TYPE csp_transfer_upstacker_phase_status_enum :
(		
	CSP_TRANSFER_UPSTACKER_STATUS_PHASE_START								:= 0,
	CSP_TRANSFER_UPSTACKER_STATUS_PHASE_CHECK_VM_STATUS						:= 1,
	CSP_TRANSFER_UPSTACKER_STATUS_PHASE_GET_VM_POS							:= 2,
	CSP_TRANSFER_UPSTACKER_STATUS_PHASE_CALCULATE_SLAVE_POS					:= 3,
	CSP_TRANSFER_UPSTACKER_STATUS_PHASE_CALCULATE_SLAVE_DOWN_POS			:= 600,
	CSP_TRANSFER_UPSTACKER_STATUS_PHASE_CHECK_CALCULATED_SLAVE_DOWN_POS		:= 601,
	CSP_TRANSFER_UPSTACKER_STATUS_PHASE_CALCULATE_SLAVE_UP_POS				:= 602,
	CSP_TRANSFER_UPSTACKER_STATUS_PHASE_CHECK_CALCULATED_SLAVE_UP_POS		:= 603,
	CSP_TRANSFER_UPSTACKER_STATUS_PHASE_CALCULATE_SLAVE_LS_FINGER_POS		:= 604,
	CSP_TRANSFER_UPSTACKER_STATUS_PHASE_CHECK_CALCULATED_SLAVE_LSFINGR_POS	:= 605,
	CSP_TRANSFER_UPSTACKER_STATUS_PHASE_CALCULATE_SLAVE_OS_FINGER_POS		:= 606,
	CSP_TRANSFER_UPSTACKER_STATUS_PHASE_CHECK_CALCULATED_SLAVE_OSFINGR_POS	:= 607,
	CSP_TRANSFER_UPSTACKER_STATUS_PHASE_CHECK_SLAVE_POS						:= 4,
	CSP_TRANSFER_UPSTACKER_STATUS_PHASE_SIMPLE_MOVE_AVAILABLE				:= 5,
	CSP_TRANSFER_UPSTACKER_STATUS_PHASE_CALCULATE_IDLE_POSITION				:= 10,
	CSP_TRANSFER_UPSTACKER_STATUS_PHASE_REDEFINE_IDLE_POSITION				:= 15,
	CSP_TRANSFER_UPSTACKER_STATUS_PHASE_READ_IDLE_POSITION					:= 20,
	CSP_TRANSFER_UPSTACKER_STATUS_PHASE_CALCULATE_SLAVE_POSITION			:= 30,
	CSP_TRANSFER_UPSTACKER_STATUS_PHASE_READ_SLAVE_POSITION					:= 40,
	CSP_TRANSFER_UPSTACKER_STATUS_PHASE_CALCULATE_VIRTUAL_POSITION			:= 50,
	CSP_TRANSFER_UPSTACKER_STATUS_PHASE_READ_VIRTUAL_POSITION				:= 60,
	CSP_TRANSFER_UPSTACKER_STATUS_PHASE_CHECK_CASE							:= 70,
	CSP_TRANSFER_UPSTACKER_STATUS_PHASE_DISABLE 							:= 80,
	CSP_TRANSFER_UPSTACKER_STATUS_PHASE_ENABLE 								:= 90,
	CSP_TRANSFER_UPSTACKER_STATUS_PHASE_ENABLED								:= 100,
	CSP_TRANSFER_UPSTACKER_STATUS_PHASE_CHECK_UPSTREAM_SKIP_PHASING			:= 101,
	CSP_TRANSFER_UPSTACKER_STATUS_PHASE_CHECK_DOWNSTREAM_SKIP_PHASE_1		:= 110,
	CSP_TRANSFER_UPSTACKER_STATUS_PHASE_CALCULATE_MASTER_POSITION			:= 150,
	CSP_TRANSFER_UPSTACKER_STATUS_PHASE_READ_MASTER_POSITION				:= 160,
	CSP_TRANSFER_UPSTACKER_STATUS_PHASE_ERROR_ON_MASTER_CALC				:= 161,
	CSP_TRANSFER_UPSTACKER_STATUS_PHASE_MOVE_UPSTREAM_FROM_ERROR_POS		:= 162,
	CSP_TRANSFER_UPSTACKER_STATUS_PHASE_WAIT_MOVE_DONE_UP_FROM_ERROR_POS	:= 163,
	CSP_TRANSFER_UPSTACKER_STATUS_PHASE_MOVE_DOWNSTREAM_FROM_ERROR_POS		:= 164,
	CSP_TRANSFER_UPSTACKER_STATUS_PHASE_WAIT_MOVE_DONE_DOWN_FROM_ERROR_POS	:= 165,
	CSP_TRANSFER_UPSTACKER_STATUS_PHASE_REDEFINE_MASTER_POSITION_STEP1		:= 170,
	CSP_TRANSFER_UPSTACKER_STATUS_PHASE_ENGAGE_DOWNSTREAM_STEP1				:= 180,
	CSP_TRANSFER_UPSTACKER_STATUS_PHASE_ENGAGE_UPSTREAM_STEP1				:= 190,
	CSP_TRANSFER_UPSTACKER_STATUS_PHASE_MOVE_MASTER_STEP1					:= 200,
	CSP_TRANSFER_UPSTACKER_STATUS_PHASE_DISENGAGE_STEP1						:= 210,
	CSP_TRANSFER_UPSTACKER_STATUS_PHASE_DISENGAGED_STEP1					:= 220,
	CSP_TRANSFER_UPSTACKER_STATUS_PHASE_CALCULE_DOWNSTREAM_START_POSITION_1	:= 230,
	CSP_TRANSFER_UPSTACKER_STATUS_PHASE_MOVE_DOWNSTREAM_START_POSITION_1	:= 240,
	CSP_TRANSFER_UPSTACKER_STATUS_PHASE_MOVED_DOWNSTREAM_START_POSITION_1	:= 250,
	CSP_TRANSFER_UPSTACKER_STATUS_PHASE_CALCULE_UPSTREAM_START_POSITION		:= 260,
	CSP_TRANSFER_UPSTACKER_STATUS_PHASE_MOVE_UPSTREAM_START_POSITION		:= 270,
	CSP_TRANSFER_UPSTACKER_STATUS_PHASE_MOVED_UPSTREAM_START_POSITION		:= 280,
	CSP_TRANSFER_UPSTACKER_STATUS_PHASE_CALCULE_DOWNSTREAM_START_POSITION_2	:= 281,
	CSP_TRANSFER_UPSTACKER_STATUS_PHASE_MOVE_DOWNSTREAM_START_POSITION_2	:= 282,
	CSP_TRANSFER_UPSTACKER_STATUS_PHASE_MOVED_DOWNSTREAM_START_POSITION_2	:= 283,
	CSP_TRANSFER_UPSTACKER_STATUS_PHASE_REDEFINE_MASTER_POSITION_STEP2		:= 290,
	CSP_TRANSFER_UPSTACKER_STATUS_PHASE_ENGAGE_DOWNSTREAM_STEP2				:= 300,
	CSP_TRANSFER_UPSTACKER_STATUS_PHASE_ENGAGE_UPSTREAM_STEP2				:= 310,
	CSP_TRANSFER_UPSTACKER_STATUS_PHASE_MOVE_MASTER_STEP2					:= 320,
	CSP_TRANSFER_UPSTACKER_STATUS_PHASE_DISENGAGE_STEP2						:= 330,
	CSP_TRANSFER_UPSTACKER_STATUS_PHASE_REDEFINE_MASTER_POSITION			:= 340,
	CSP_TRANSFER_UPSTACKER_STATUS_PHASE_MASTER_POSITION_REDEFINED			:= 350,
	CSP_TRANSFER_UPSTACKER_STATUS_PHASE_MOVE_PHASING						:= 400,
	CSP_TRANSFER_UPSTACKER_STATUS_PHASE_MOVED_PHASING						:= 410,	
	CSP_TRANSFER_UPSTACKER_STATUS_PHASE_CALCULATE_UPSTACKER_MASTER_POS		:= 415,	
	CSP_TRANSFER_UPSTACKER_STATUS_PHASE_CALCULATED_UPSTACKER_MASTER_POS_DONE:= 416,
	CSP_TRANSFER_UPSTACKER_STATUS_PHASE_REDFINE_MASTER_ABS_PHASE			:= 420,
	CSP_TRANSFER_UPSTACKER_STATUS_PHASE_ENGAGE_DOWNSTREAM					:= 500,
	CSP_TRANSFER_UPSTACKER_STATUS_PHASE_ENGAGE_UPSTREAM						:= 510,
	CSP_TRANSFER_UPSTACKER_STATUS_PHASE_MOVE_FINGER_LS						:= 512,
	CSP_TRANSFER_UPSTACKER_STATUS_PHASE_MOVE_FINGER_OS						:= 514,
	CSP_TRANSFER_UPSTACKER_STATUS_PHASE_ENGAGE_FINGER_LS					:= 520,
	CSP_TRANSFER_UPSTACKER_STATUS_PHASE_ENGAGE_FINGER_OS					:= 530,
	CSP_TRANSFER_UPSTACKER_STATUS_PHASE_ALL_ENGAGED							:= 540,
	CSP_TRANSFER_UPSTACKER_STATUS_PHASE_MOVE_MASTER_TO_IDLE					:= 550,
	CSP_TRANSFER_UPSTACKER_STATUS_PHASE_MOVED_MASTER_TO_IDLE				:= 560,
	CSP_TRANSFER_UPSTACKER_STATUS_PHASE_DONE 								:= 900,
	CSP_TRANSFER_UPSTACKER_STATUS_PHASE_ERROR 								:= 999
) := CSP_TRANSFER_UPSTACKER_STATUS_PHASE_START;
END_TYPE

(* stored: Version 1.1.0.1, ProductVersion 3.1.4024.3
   DUT csp_transfer_upstacker_phase_status_enum: Id {8adfbc8c-09aa-43e0-897e-a70f9b8bfeaa} *)
